// TwinCAT 3 PLC project PLC
// Title: TcUnits
// Author: Roald Ruiter
// ProjectVersion: 0.1.0
// Description: Aliases for units
// ProgramVersion: 3.1.4023.0
// libraries:
//   Tc2_Standard, * (Beckhoff Automation GmbH)
//   Tc2_System, * (Beckhoff Automation GmbH)
//   Tc3_Module, * (Beckhoff Automation GmbH)
// project tree:
//   Distance/ Millimeter.TcDUT (not stored)
//   Force/ Newton.TcDUT
//   / Percent.TcDUT (not stored)
//   Speed/ MillimeterPerSecond.TcDUT
//   Time/ Millisecond.TcDUT (not stored)
//   Torque/ NewtonMeter.TcDUT (not stored)
//   Weight/ Kilogram.TcDUT

// ---- Force/Newton.TcDUT
TYPE Newton : LREAL;
END_TYPE

// ---- Speed/MillimeterPerSecond.TcDUT
TYPE MillimeterPerSecond : LREAL;
END_TYPE

// ---- Weight/Kilogram.TcDUT
TYPE Kilogram : LREAL;
END_TYPE
